FUNCTION_BLOCK PUBLIC FB_AirConComfortCommand IMPLEMENTS I_Command
VAR
	refAirConditioning : REFERENCE TO FB_AirConditioning;
END_VAR

METHOD Execute
IF (__ISVALIDREF(THIS^.refAirConditioning)) THEN
	THIS^.refAirConditioning.Activate();
	THIS^.refAirConditioning.SetTemperature(20.0);
END_IF
END_METHOD

METHOD FB_init : BOOL
VAR_INPUT
	bInitRetains : BOOL; // if TRUE, the retain variables are initialized (warm start / cold start)
	bInCopyCode : BOOL;  // if TRUE, the instance afterwards gets moved into the copy code (online change)
	refAirConditioning : REFERENCE TO FB_AirConditioning;
END_VAR
IF (__ISVALIDREF(refAirConditioning)) THEN
	THIS^.refAirConditioning REF= refAirConditioning;
ELSE
	THIS^.refAirConditioning REF= 0;
END_IF
END_METHOD

METHOD Undo
IF (__ISVALIDREF(THIS^.refAirConditioning)) THEN
	THIS^.refAirConditioning.Activate();
	THIS^.refAirConditioning.SetTemperature(17.5);
END_IF
END_METHOD

END_FUNCTION_BLOCK

(* stored: Version 1.1.0.1, ProductVersion 3.1.4020.3
   POU FB_AirConComfortCommand: Id {fa70c319-e680-4f43-bf75-6b04781fe123}, SpecialFunc None
   Method Execute: Id {0530f813-4259-4fee-8d29-4203989fd02f}
   Method FB_init: Id {4d0f061f-23e5-4b59-87d0-78ae1b8327c5}
   Method Undo: Id {03366f51-978b-46b0-b8c2-87489b0e9e31} *)
